TYPE ST_Unit :
STRUCT
	eType		: E_Unit;
	iHitPoint	: INT;
	iProgress	: INT;
END_STRUCT
END_TYPE

(* stored: Version 1.1.0.1, ProductVersion 3.1.4024.12
   DUT ST_Unit: Id {235696af-b39b-4ff8-94af-779fe1d66eb9} *)
